FUNCTION_BLOCK EventLogger
VAR
	EventBuffer : ARRAY[1..MAXIMUM_SIZE_OF_EVENT_BUFFER] OF ST_Event;
	CurrentEventBufferIndex : INT := 0;
	_PersistentEventLogger : I_PersistentEventStorage; // (2) store the reference to interface locally in FB
END_VAR
VAR CONSTANT
	MAXIMUM_SIZE_OF_EVENT_BUFFER : INT := 100;
END_VAR

// Returns True if Add was successful and False if the buffer is full
METHOD PUBLIC AddEvent : BOOL
VAR_INPUT
	eEventType : E_EventType;
	eEventSeverity : TcEventSeverity;
	nEventIdentity : UDINT;
	sEventText : STRING(255);
END_VAR
IF NOT IsEventBufferFull() THEN
	CurrentEventBufferIndex := CurrentEventBufferIndex + 1;
	EventBuffer[CurrentEventBufferIndex].eEventType := eEventType;
	EventBuffer[CurrentEventBufferIndex].eEventSeverity := eEventSeverity;
	EventBuffer[CurrentEventBufferIndex].nEventIdentity := nEventIdentity;
	EventBuffer[CurrentEventBufferIndex].sEventText := sEventText;
	UpdateEventTimestampWithSystemTime(stEvent := EventBuffer[CurrentEventBufferIndex]); 
// this function will take a reference to this buffer location and update dtTimastamp of Event
	AddEvent := TRUE;
ELSE
	AddEvent := FALSE;
END_IF
// Here we want to store our Events persistently
_PersistentEventLogger.StoreEvent(stEvent := EventBuffer[CurrentEventBufferIndex]);
END_METHOD

METHOD FB_init : BOOL
VAR_INPUT
	bInitRetains : BOOL; // if TRUE, the retain variables are initialized (warm start / cold start)
	bInCopyCode : BOOL;  // if TRUE, the instance afterwards gets moved into the copy code (online change)
	iPersitentEventStorage : I_PersistentEventStorage; // (1) reference to the interface
END_VAR
_PersistentEventLogger := iPersitentEventStorage; // (3)
END_METHOD

METHOD PRIVATE IsEventBufferFull : BOOL
IF (CurrentEventBufferIndex + 1) > MAXIMUM_SIZE_OF_EVENT_BUFFER THEN
	IsEventBufferFull := TRUE;
ELSE
	IsEventBufferFull := FALSE;
END_IF
END_METHOD

END_FUNCTION_BLOCK

(* stored: Version 1.1.0.1, ProductVersion 3.1.4024.12
   POU EventLogger: Id {08cbf15c-8688-4dd9-ab6b-e1a448de205a}, SpecialFunc None
   Method AddEvent: Id {e49f4b21-dfc7-438e-a953-7966645755e4}
   Method FB_init: Id {6cf4241f-932f-4b8b-b3cc-1e543ad81590}
   Method IsEventBufferFull: Id {2b2e068d-0933-4786-8ed4-5fa954dc4519} *)
